// TIA Portal V15.1 export
// export: Created 2024-06-21T08:41:24.7337865Z, ExportSetting WithDefaults, DisplayName Totally Integrated Automation Portal, DisplayVersion V15.1 Update 5, DisplayName TIA Portal Openness, DisplayVersion V15.1 Update 5, DisplayName SINAMICS Startdrive Advanced, DisplayVersion V15.1, DisplayName G130, G150, S120, S150, SINAMICS MV, S210, DisplayVersion V15.1, DisplayName G110M, G120, G120C, G120D, G120P, DisplayVersion V15.1, DisplayName STEP 7 Professional, DisplayVersion V15.1 Update 5, DisplayName STEP 7 Safety, DisplayVersion V15.1, DisplayName WinCC Professional, DisplayVersion V15.1 Update 5, DisplayName SIMATIC Visualization Architect, DisplayVersion V15.1
FUNCTION "209230ZM01Modes" : Void   // FC401, FBD
TITLE = 209230ZM01 Modes
{ S7_Optimized_Access := 'FALSE' }
AUTHOR : VCC
FAMILY : Local
NAME : Local
VERSION : 0.1
// stored: AutoNumber false, IsIECCheckEnabled false, SetENOAutomatically False, UDAEnableTagReadback false
   VAR_OUTPUT
      O_AlarmA : Bool;   // Alarm A
      O_AlarmB : Bool;   // Alarm B
      O_AlarmC : Bool;   // Alarm C
      O_AlarmD : Bool;   // Alarm D
      O_AlarmABCondition : Bool;   // Alarms resetable
   END_VAR
   VAR_TEMP
      NotUsed : Bool;
   END_VAR
BEGIN

REGION Network 1: **** 1 - Inputs **** General Functions
   // General Functions
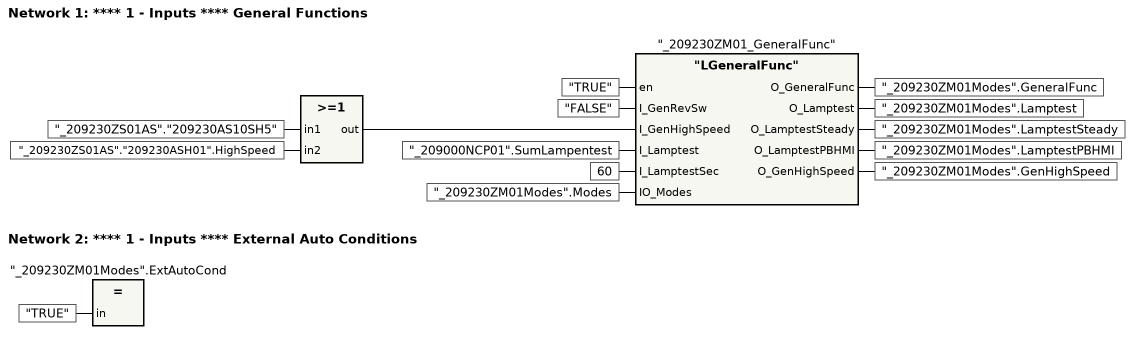
   IF "TRUE" THEN
       "_209230ZM01_GeneralFunc"(I_GenRevSw := "FALSE",   // "LGeneralFunc"
                               I_GenHighSpeed := "_209230ZS01AS"."209230AS10SH5" OR "_209230ZS01AS"."209230ASH01".HighSpeed,
                               I_Lamptest := "_209000NCP01".SumLampentest,
                               I_LamptestSec := 60,
                               IO_Modes := "_209230ZM01Modes".Modes,
                               O_GeneralFunc => "_209230ZM01Modes".GeneralFunc,
                               O_Lamptest => "_209230ZM01Modes".Lamptest,
                               O_LamptestSteady => "_209230ZM01Modes".LamptestSteady,
                               O_LamptestPBHMI => "_209230ZM01Modes".LamptestPBHMI,
                               O_GenHighSpeed => "_209230ZM01Modes".GenHighSpeed);
   END_IF;
END_REGION

REGION Network 2: **** 1 - Inputs **** External Auto Conditions
   "_209230ZM01Modes".ExtAutoCond := "TRUE";
END_REGION

REGION Network 3: **** 4.5 - Machine Status - Modes **** Mode selector
   // Mode selector
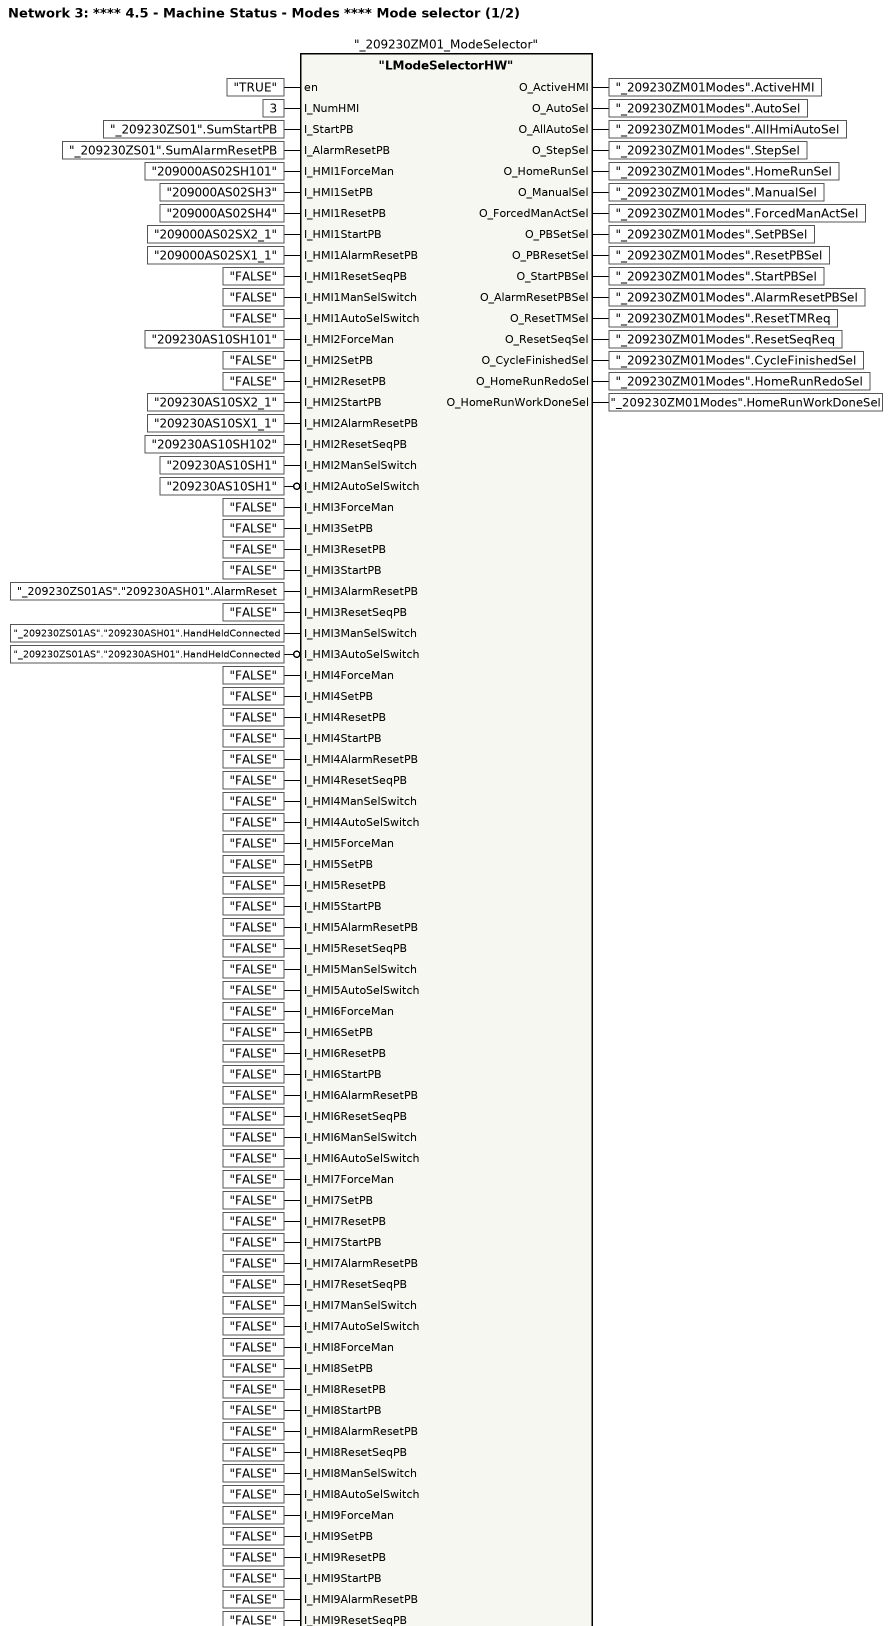
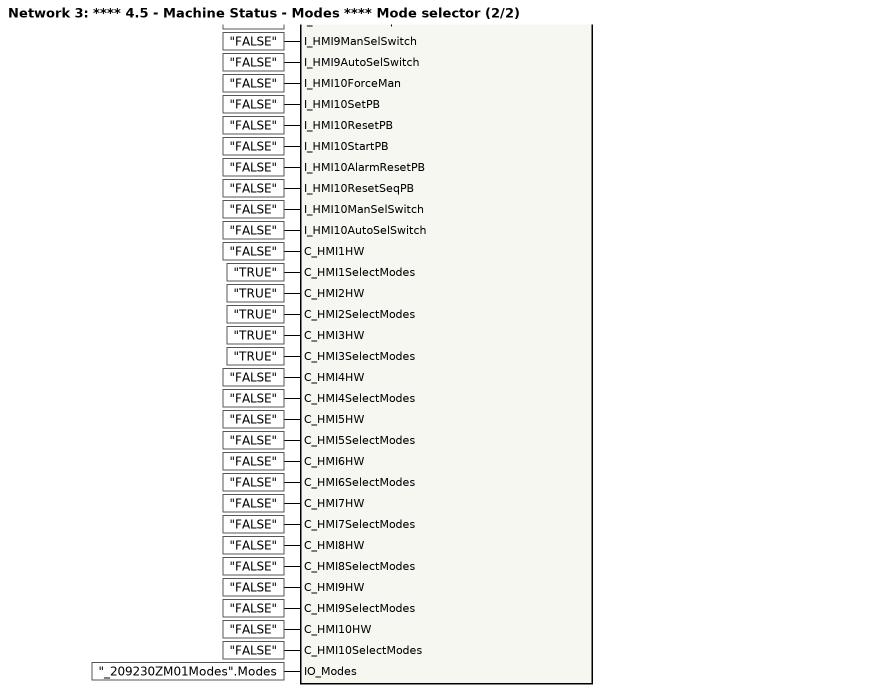
   IF "TRUE" THEN
       "_209230ZM01_ModeSelector"(I_NumHMI := 3,   // "LModeSelectorHW"
                               I_StartPB := "_209230ZS01".SumStartPB,
                               I_AlarmResetPB := "_209230ZS01".SumAlarmResetPB,
                               I_HMI1ForceMan := "209000AS02SH101",
                               I_HMI1SetPB := "209000AS02SH3",
                               I_HMI1ResetPB := "209000AS02SH4",
                               I_HMI1StartPB := "209000AS02SX2_1",
                               I_HMI1AlarmResetPB := "209000AS02SX1_1",
                               I_HMI1ResetSeqPB := "FALSE",
                               I_HMI1ManSelSwitch := "FALSE",
                               I_HMI1AutoSelSwitch := "FALSE",
                               I_HMI2ForceMan := "209230AS10SH101",
                               I_HMI2SetPB := "FALSE",
                               I_HMI2ResetPB := "FALSE",
                               I_HMI2StartPB := "209230AS10SX2_1",
                               I_HMI2AlarmResetPB := "209230AS10SX1_1",
                               I_HMI2ResetSeqPB := "209230AS10SH102",
                               I_HMI2ManSelSwitch := "209230AS10SH1",
                               I_HMI2AutoSelSwitch := NOT "209230AS10SH1",
                               I_HMI3ForceMan := "FALSE",
                               I_HMI3SetPB := "FALSE",
                               I_HMI3ResetPB := "FALSE",
                               I_HMI3StartPB := "FALSE",
                               I_HMI3AlarmResetPB := "_209230ZS01AS"."209230ASH01".AlarmReset,
                               I_HMI3ResetSeqPB := "FALSE",
                               I_HMI3ManSelSwitch := "_209230ZS01AS"."209230ASH01".HandHeldConnected,
                               I_HMI3AutoSelSwitch := NOT "_209230ZS01AS"."209230ASH01".HandHeldConnected,
                               I_HMI4ForceMan := "FALSE",
                               I_HMI4SetPB := "FALSE",
                               I_HMI4ResetPB := "FALSE",
                               I_HMI4StartPB := "FALSE",
                               I_HMI4AlarmResetPB := "FALSE",
                               I_HMI4ResetSeqPB := "FALSE",
                               I_HMI4ManSelSwitch := "FALSE",
                               I_HMI4AutoSelSwitch := "FALSE",
                               I_HMI5ForceMan := "FALSE",
                               I_HMI5SetPB := "FALSE",
                               I_HMI5ResetPB := "FALSE",
                               I_HMI5StartPB := "FALSE",
                               I_HMI5AlarmResetPB := "FALSE",
                               I_HMI5ResetSeqPB := "FALSE",
                               I_HMI5ManSelSwitch := "FALSE",
                               I_HMI5AutoSelSwitch := "FALSE",
                               I_HMI6ForceMan := "FALSE",
                               I_HMI6SetPB := "FALSE",
                               I_HMI6ResetPB := "FALSE",
                               I_HMI6StartPB := "FALSE",
                               I_HMI6AlarmResetPB := "FALSE",
                               I_HMI6ResetSeqPB := "FALSE",
                               I_HMI6ManSelSwitch := "FALSE",
                               I_HMI6AutoSelSwitch := "FALSE",
                               I_HMI7ForceMan := "FALSE",
                               I_HMI7SetPB := "FALSE",
                               I_HMI7ResetPB := "FALSE",
                               I_HMI7StartPB := "FALSE",
                               I_HMI7AlarmResetPB := "FALSE",
                               I_HMI7ResetSeqPB := "FALSE",
                               I_HMI7ManSelSwitch := "FALSE",
                               I_HMI7AutoSelSwitch := "FALSE",
                               I_HMI8ForceMan := "FALSE",
                               I_HMI8SetPB := "FALSE",
                               I_HMI8ResetPB := "FALSE",
                               I_HMI8StartPB := "FALSE",
                               I_HMI8AlarmResetPB := "FALSE",
                               I_HMI8ResetSeqPB := "FALSE",
                               I_HMI8ManSelSwitch := "FALSE",
                               I_HMI8AutoSelSwitch := "FALSE",
                               I_HMI9ForceMan := "FALSE",
                               I_HMI9SetPB := "FALSE",
                               I_HMI9ResetPB := "FALSE",
                               I_HMI9StartPB := "FALSE",
                               I_HMI9AlarmResetPB := "FALSE",
                               I_HMI9ResetSeqPB := "FALSE",
                               I_HMI9ManSelSwitch := "FALSE",
                               I_HMI9AutoSelSwitch := "FALSE",
                               I_HMI10ForceMan := "FALSE",
                               I_HMI10SetPB := "FALSE",
                               I_HMI10ResetPB := "FALSE",
                               I_HMI10StartPB := "FALSE",
                               I_HMI10AlarmResetPB := "FALSE",
                               I_HMI10ResetSeqPB := "FALSE",
                               I_HMI10ManSelSwitch := "FALSE",
                               I_HMI10AutoSelSwitch := "FALSE",
                               C_HMI1HW := "FALSE",
                               C_HMI1SelectModes := "TRUE",
                               C_HMI2HW := "TRUE",
                               C_HMI2SelectModes := "TRUE",
                               C_HMI3HW := "TRUE",
                               C_HMI3SelectModes := "TRUE",
                               C_HMI4HW := "FALSE",
                               C_HMI4SelectModes := "FALSE",
                               C_HMI5HW := "FALSE",
                               C_HMI5SelectModes := "FALSE",
                               C_HMI6HW := "FALSE",
                               C_HMI6SelectModes := "FALSE",
                               C_HMI7HW := "FALSE",
                               C_HMI7SelectModes := "FALSE",
                               C_HMI8HW := "FALSE",
                               C_HMI8SelectModes := "FALSE",
                               C_HMI9HW := "FALSE",
                               C_HMI9SelectModes := "FALSE",
                               C_HMI10HW := "FALSE",
                               C_HMI10SelectModes := "FALSE",
                               IO_Modes := "_209230ZM01Modes".Modes,
                               O_ActiveHMI => "_209230ZM01Modes".ActiveHMI,
                               O_AutoSel => "_209230ZM01Modes".AutoSel,
                               O_AllAutoSel => "_209230ZM01Modes".AllHmiAutoSel,
                               O_StepSel => "_209230ZM01Modes".StepSel,
                               O_HomeRunSel => "_209230ZM01Modes".HomeRunSel,
                               O_ManualSel => "_209230ZM01Modes".ManualSel,
                               O_ForcedManActSel => "_209230ZM01Modes".ForcedManActSel,
                               O_PBSetSel => "_209230ZM01Modes".SetPBSel,
                               O_PBResetSel => "_209230ZM01Modes".ResetPBSel,
                               O_StartPBSel => "_209230ZM01Modes".StartPBSel,
                               O_AlarmResetPBSel => "_209230ZM01Modes".AlarmResetPBSel,
                               O_ResetTMSel => "_209230ZM01Modes".ResetTMReq,
                               O_ResetSeqSel => "_209230ZM01Modes".ResetSeqReq,
                               O_CycleFinishedSel => "_209230ZM01Modes".CycleFinishedSel,
                               O_HomeRunRedoSel => "_209230ZM01Modes".HomeRunRedoSel,
                               O_HomeRunWorkDoneSel => "_209230ZM01Modes".HomeRunWorkDoneSel);
   END_IF;
END_REGION

REGION Network 4: **** 4.5 - Machine Status - Modes **** Modes
   // Modes
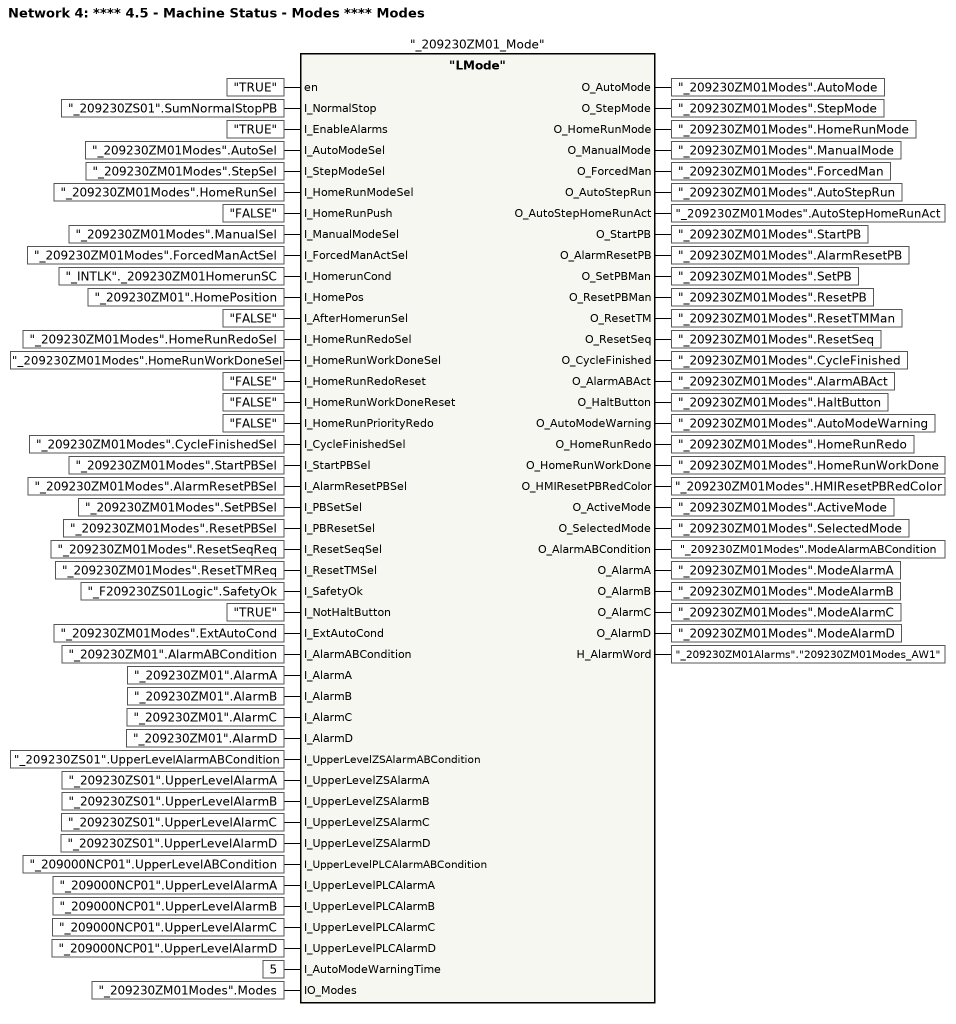
   IF "TRUE" THEN
       "_209230ZM01_Mode"(I_NormalStop := "_209230ZS01".SumNormalStopPB,   // "LMode"
                          I_EnableAlarms := "TRUE",
                          I_AutoModeSel := "_209230ZM01Modes".AutoSel,
                          I_StepModeSel := "_209230ZM01Modes".StepSel,
                          I_HomeRunModeSel := "_209230ZM01Modes".HomeRunSel,
                          I_HomeRunPush := "FALSE",
                          I_ManualModeSel := "_209230ZM01Modes".ManualSel,
                          I_ForcedManActSel := "_209230ZM01Modes".ForcedManActSel,
                          I_HomerunCond := "_INTLK"._209230ZM01HomerunSC,
                          I_HomePos := "_209230ZM01".HomePosition,
                          I_AfterHomerunSel := "FALSE",
                          I_HomeRunRedoSel := "_209230ZM01Modes".HomeRunRedoSel,
                          I_HomeRunWorkDoneSel := "_209230ZM01Modes".HomeRunWorkDoneSel,
                          I_HomeRunRedoReset := "FALSE",
                          I_HomeRunWorkDoneReset := "FALSE",
                          I_HomeRunPriorityRedo := "FALSE",
                          I_CycleFinishedSel := "_209230ZM01Modes".CycleFinishedSel,
                          I_StartPBSel := "_209230ZM01Modes".StartPBSel,
                          I_AlarmResetPBSel := "_209230ZM01Modes".AlarmResetPBSel,
                          I_PBSetSel := "_209230ZM01Modes".SetPBSel,
                          I_PBResetSel := "_209230ZM01Modes".ResetPBSel,
                          I_ResetSeqSel := "_209230ZM01Modes".ResetSeqReq,
                          I_ResetTMSel := "_209230ZM01Modes".ResetTMReq,
                          I_SafetyOk := "_F209230ZS01Logic".SafetyOk,
                          I_NotHaltButton := "TRUE",
                          I_ExtAutoCond := "_209230ZM01Modes".ExtAutoCond,
                          I_AlarmABCondition := "_209230ZM01".AlarmABCondition,
                          I_AlarmA := "_209230ZM01".AlarmA,
                          I_AlarmB := "_209230ZM01".AlarmB,
                          I_AlarmC := "_209230ZM01".AlarmC,
                          I_AlarmD := "_209230ZM01".AlarmD,
                          I_UpperLevelZSAlarmABCondition := "_209230ZS01".UpperLevelAlarmABCondition,
                          I_UpperLevelZSAlarmA := "_209230ZS01".UpperLevelAlarmA,
                          I_UpperLevelZSAlarmB := "_209230ZS01".UpperLevelAlarmB,
                          I_UpperLevelZSAlarmC := "_209230ZS01".UpperLevelAlarmC,
                          I_UpperLevelZSAlarmD := "_209230ZS01".UpperLevelAlarmD,
                          I_UpperLevelPLCAlarmABCondition := "_209000NCP01".UpperLevelABCondition,
                          I_UpperLevelPLCAlarmA := "_209000NCP01".UpperLevelAlarmA,
                          I_UpperLevelPLCAlarmB := "_209000NCP01".UpperLevelAlarmB,
                          I_UpperLevelPLCAlarmC := "_209000NCP01".UpperLevelAlarmC,
                          I_UpperLevelPLCAlarmD := "_209000NCP01".UpperLevelAlarmD,
                          I_AutoModeWarningTime := 5,
                          IO_Modes := "_209230ZM01Modes".Modes,
                          O_AutoMode => "_209230ZM01Modes".AutoMode,
                          O_StepMode => "_209230ZM01Modes".StepMode,
                          O_HomeRunMode => "_209230ZM01Modes".HomeRunMode,
                          O_ManualMode => "_209230ZM01Modes".ManualMode,
                          O_ForcedMan => "_209230ZM01Modes".ForcedMan,
                          O_AutoStepRun => "_209230ZM01Modes".AutoStepRun,
                          O_AutoStepHomeRunAct => "_209230ZM01Modes".AutoStepHomeRunAct,
                          O_StartPB => "_209230ZM01Modes".StartPB,
                          O_AlarmResetPB => "_209230ZM01Modes".AlarmResetPB,
                          O_SetPBMan => "_209230ZM01Modes".SetPB,
                          O_ResetPBMan => "_209230ZM01Modes".ResetPB,
                          O_ResetTM => "_209230ZM01Modes".ResetTMMan,
                          O_ResetSeq => "_209230ZM01Modes".ResetSeq,
                          O_CycleFinished => "_209230ZM01Modes".CycleFinished,
                          O_AlarmABAct => "_209230ZM01Modes".AlarmABAct,
                          O_HaltButton => "_209230ZM01Modes".HaltButton,
                          O_AutoModeWarning => "_209230ZM01Modes".AutoModeWarning,
                          O_HomeRunRedo => "_209230ZM01Modes".HomeRunRedo,
                          O_HomeRunWorkDone => "_209230ZM01Modes".HomeRunWorkDone,
                          O_HMIResetPBRedColor => "_209230ZM01Modes".HMIResetPBRedColor,
                          O_ActiveMode => "_209230ZM01Modes".ActiveMode,
                          O_SelectedMode => "_209230ZM01Modes".SelectedMode,
                          O_AlarmABCondition => "_209230ZM01Modes".ModeAlarmABCondition,
                          O_AlarmA => "_209230ZM01Modes".ModeAlarmA,
                          O_AlarmB => "_209230ZM01Modes".ModeAlarmB,
                          O_AlarmC => "_209230ZM01Modes".ModeAlarmC,
                          O_AlarmD => "_209230ZM01Modes".ModeAlarmD,
                          H_AlarmWord => "_209230ZM01Alarms"."209230ZM01Modes_AW1");
   END_IF;
END_REGION

REGION Network 5: **** 4.5 - Machine Status - Modes **** Production Modes
   // Production Modes
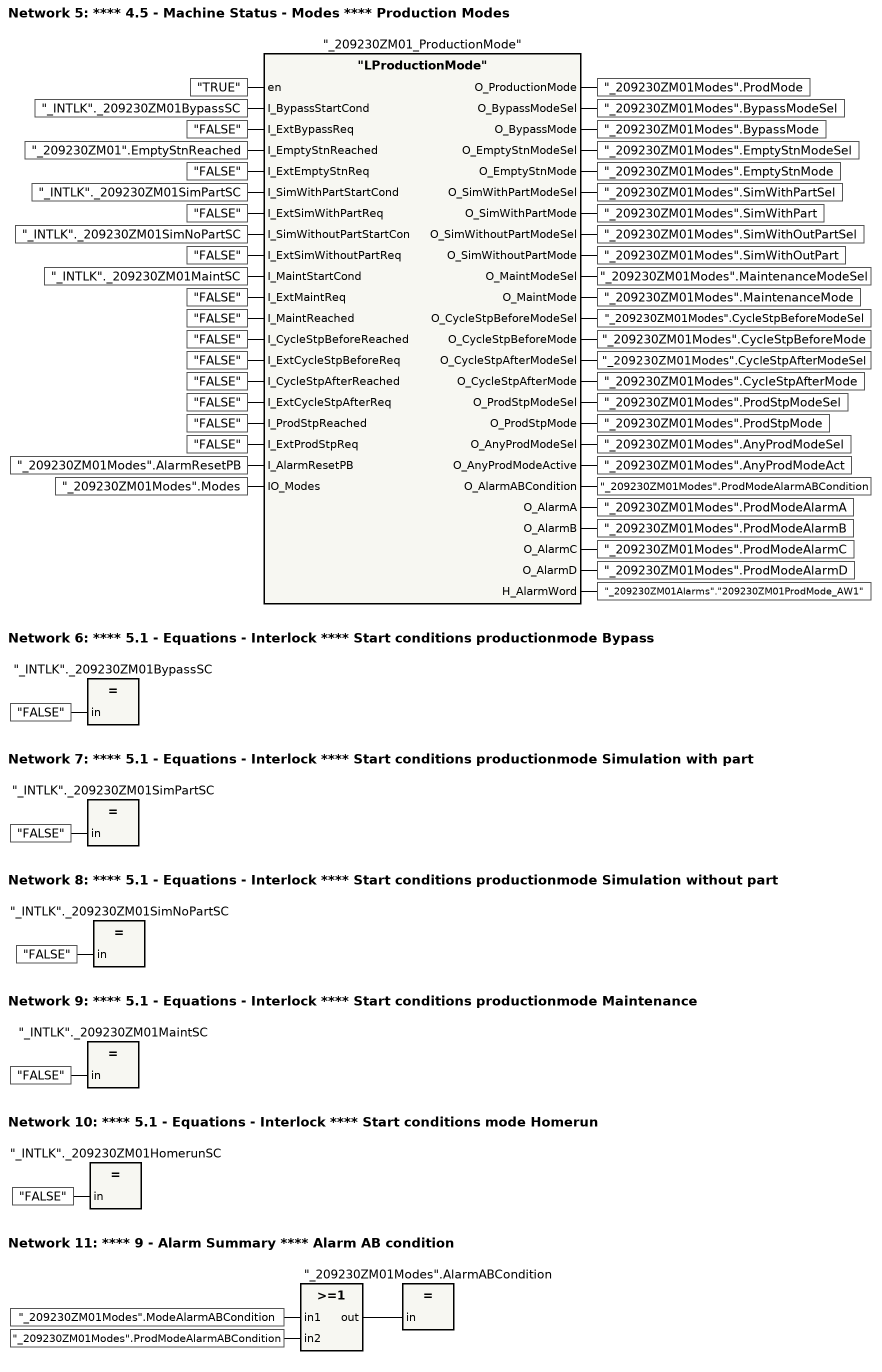
   IF "TRUE" THEN
       "_209230ZM01_ProductionMode"(I_BypassStartCond := "_INTLK"._209230ZM01BypassSC,   // "LProductionMode"
                               I_ExtBypassReq := "FALSE",
                               I_EmptyStnReached := "_209230ZM01".EmptyStnReached,
                               I_ExtEmptyStnReq := "FALSE",
                               I_SimWithPartStartCond := "_INTLK"._209230ZM01SimPartSC,
                               I_ExtSimWithPartReq := "FALSE",
                               I_SimWithoutPartStartCon := "_INTLK"._209230ZM01SimNoPartSC,
                               I_ExtSimWithoutPartReq := "FALSE",
                               I_MaintStartCond := "_INTLK"._209230ZM01MaintSC,
                               I_ExtMaintReq := "FALSE",
                               I_MaintReached := "FALSE",
                               I_CycleStpBeforeReached := "FALSE",
                               I_ExtCycleStpBeforeReq := "FALSE",
                               I_CycleStpAfterReached := "FALSE",
                               I_ExtCycleStpAfterReq := "FALSE",
                               I_ProdStpReached := "FALSE",
                               I_ExtProdStpReq := "FALSE",
                               I_AlarmResetPB := "_209230ZM01Modes".AlarmResetPB,
                               IO_Modes := "_209230ZM01Modes".Modes,
                               O_ProductionMode => "_209230ZM01Modes".ProdMode,
                               O_BypassModeSel => "_209230ZM01Modes".BypassModeSel,
                               O_BypassMode => "_209230ZM01Modes".BypassMode,
                               O_EmptyStnModeSel => "_209230ZM01Modes".EmptyStnModeSel,
                               O_EmptyStnMode => "_209230ZM01Modes".EmptyStnMode,
                               O_SimWithPartModeSel => "_209230ZM01Modes".SimWithPartSel,
                               O_SimWithPartMode => "_209230ZM01Modes".SimWithPart,
                               O_SimWithoutPartModeSel => "_209230ZM01Modes".SimWithOutPartSel,
                               O_SimWithoutPartMode => "_209230ZM01Modes".SimWithOutPart,
                               O_MaintModeSel => "_209230ZM01Modes".MaintenanceModeSel,
                               O_MaintMode => "_209230ZM01Modes".MaintenanceMode,
                               O_CycleStpBeforeModeSel => "_209230ZM01Modes".CycleStpBeforeModeSel,
                               O_CycleStpBeforeMode => "_209230ZM01Modes".CycleStpBeforeMode,
                               O_CycleStpAfterModeSel => "_209230ZM01Modes".CycleStpAfterModeSel,
                               O_CycleStpAfterMode => "_209230ZM01Modes".CycleStpAfterMode,
                               O_ProdStpModeSel => "_209230ZM01Modes".ProdStpModeSel,
                               O_ProdStpMode => "_209230ZM01Modes".ProdStpMode,
                               O_AnyProdModeSel => "_209230ZM01Modes".AnyProdModeSel,
                               O_AnyProdModeActive => "_209230ZM01Modes".AnyProdModeAct,
                               O_AlarmABCondition => "_209230ZM01Modes".ProdModeAlarmABCondition,
                               O_AlarmA => "_209230ZM01Modes".ProdModeAlarmA,
                               O_AlarmB => "_209230ZM01Modes".ProdModeAlarmB,
                               O_AlarmC => "_209230ZM01Modes".ProdModeAlarmC,
                               O_AlarmD => "_209230ZM01Modes".ProdModeAlarmD,
                               H_AlarmWord => "_209230ZM01Alarms"."209230ZM01ProdMode_AW1");
   END_IF;
END_REGION

REGION Network 6: **** 5.1 - Equations - Interlock **** Start conditions productionmode Bypass
   // Start conditions productionmode
   // Bypass
   "_INTLK"._209230ZM01BypassSC := "FALSE";
END_REGION

REGION Network 7: **** 5.1 - Equations - Interlock **** Start conditions productionmode Simulation with part
   // Start conditions productionmode
   // Simulation with part
   "_INTLK"._209230ZM01SimPartSC := "FALSE";
END_REGION

REGION Network 8: **** 5.1 - Equations - Interlock **** Start conditions productionmode Simulation without part
   // Start conditions productionmode
   // Simulation without part
   "_INTLK"._209230ZM01SimNoPartSC := "FALSE";
END_REGION

REGION Network 9: **** 5.1 - Equations - Interlock **** Start conditions productionmode Maintenance
   // Start conditions productionmode
   // Maintenance
   "_INTLK"._209230ZM01MaintSC := "FALSE";
END_REGION

REGION Network 10: **** 5.1 - Equations - Interlock **** Start conditions mode Homerun
   // Start conditions mode
   // Homerun
   "_INTLK"._209230ZM01HomerunSC := "FALSE";
END_REGION

REGION Network 11: **** 9 - Alarm Summary **** Alarm AB condition
   // Alarm AB condition
   "_209230ZM01Modes".AlarmABCondition := "_209230ZM01Modes".ModeAlarmABCondition OR "_209230ZM01Modes".ProdModeAlarmABCondition;
END_REGION

REGION Network 12: **** 9 - Alarm Summary **** Alarm A
   // Summary of alarms A
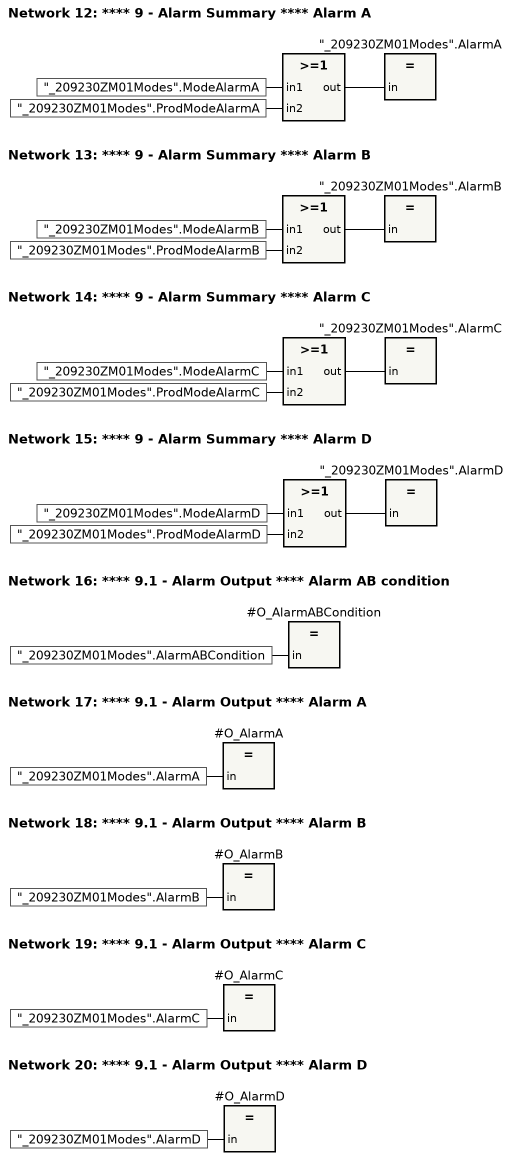
   "_209230ZM01Modes".AlarmA := "_209230ZM01Modes".ModeAlarmA OR "_209230ZM01Modes".ProdModeAlarmA;
END_REGION

REGION Network 13: **** 9 - Alarm Summary **** Alarm B
   // Summary of alarms B
   "_209230ZM01Modes".AlarmB := "_209230ZM01Modes".ModeAlarmB OR "_209230ZM01Modes".ProdModeAlarmB;
END_REGION

REGION Network 14: **** 9 - Alarm Summary **** Alarm C
   // Summary of alarms C
   "_209230ZM01Modes".AlarmC := "_209230ZM01Modes".ModeAlarmC OR "_209230ZM01Modes".ProdModeAlarmC;
END_REGION

REGION Network 15: **** 9 - Alarm Summary **** Alarm D
   // Summary of alarms D
   "_209230ZM01Modes".AlarmD := "_209230ZM01Modes".ModeAlarmD OR "_209230ZM01Modes".ProdModeAlarmD;
END_REGION

REGION Network 16: **** 9.1 - Alarm Output **** Alarm AB condition
   // Alarm AB condition
   #O_AlarmABCondition := "_209230ZM01Modes".AlarmABCondition;
END_REGION

REGION Network 17: **** 9.1 - Alarm Output **** Alarm A
   // Summary of alarms A
   #O_AlarmA := "_209230ZM01Modes".AlarmA;
END_REGION

REGION Network 18: **** 9.1 - Alarm Output **** Alarm B
   // Summary of alarms B
   #O_AlarmB := "_209230ZM01Modes".AlarmB;
END_REGION

REGION Network 19: **** 9.1 - Alarm Output **** Alarm C
   // Summary of alarms C
   #O_AlarmC := "_209230ZM01Modes".AlarmC;
END_REGION

REGION Network 20: **** 9.1 - Alarm Output **** Alarm D
   // Summary of alarms D
   #O_AlarmD := "_209230ZM01Modes".AlarmD;
END_REGION
END_FUNCTION
